  [5980] = {x=869.314, y=-99.781, z=66, rx=180, rz=144.218, shoulder=lefty, elbow=epositive, wrist=wpositive, fatherId=fReference[0]}
  [5981] = {x=870.574, y=-98.873, z=66, rx=180, rz=144.172, shoulder=lefty, elbow=epositive, wrist=wpositive, fatherId=fReference[0]}
  [5982] = {x=871.834, y=-97.963, z=66, rx=-180, rz=144.126, shoulder=lefty, elbow=epositive, wrist=wpositive, fatherId=fReference[0]}
  [5983] = {x=873.094, y=-97.052, z=66, rx=-180, rz=144.08, shoulder=lefty, elbow=epositive, wrist=wpositive, fatherId=fReference[0]}
  [5984] = {x=874.353, y=-96.14, z=66, rx=180, rz=144.036, shoulder=lefty, elbow=epositive, wrist=wpositive, fatherId=fReference[0]}
  [5985] = {x=875.611, y=-95.227, z=66, rx=-180, rz=143.991, shoulder=lefty, elbow=epositive, wrist=wpositive, fatherId=fReference[0]}
  [5986] = {x=876.869, y=-94.313, z=66, rx=180, rz=143.947, shoulder=lefty, elbow=epositive, wrist=wpositive, fatherId=fReference[0]}
  [5987] = {x=878.127, y=-93.397, z=66, rx=180, rz=143.904, shoulder=lefty, elbow=epositive, wrist=wpositive, fatherId=fReference[0]}
  [5988] = {x=879.384, y=-92.481, z=66, rx=180, rz=143.861, shoulder=lefty, elbow=epositive, wrist=wpositive, fatherId=fReference[0]}
  [5989] = {x=880.641, y=-91.563, z=66, rx=-180, rz=143.819, shoulder=lefty, elbow=epositive, wrist=wpositive, fatherId=fReference[0]}
  [5990] = {x=881.897, y=-90.644, z=66, rx=180, rz=143.777, shoulder=lefty, elbow=epositive, wrist=wpositive, fatherId=fReference[0]}
  [5991] = {x=883.153, y=-89.724, z=66, rx=-180, rz=143.735, shoulder=lefty, elbow=epositive, wrist=wpositive, fatherId=fReference[0]}
  [5992] = {x=884.409, y=-88.803, z=66, rx=-180, rz=143.694, shoulder=lefty, elbow=epositive, wrist=wpositive, fatherId=fReference[0]}
  [5993] = {x=885.664, y=-87.881, z=66, rx=-180, rz=143.654, shoulder=lefty, elbow=epositive, wrist=wpositive, fatherId=fReference[0]}
  [5994] = {x=886.919, y=-86.957, z=66, rx=180, rz=143.614, shoulder=lefty, elbow=epositive, wrist=wpositive, fatherId=fReference[0]}
  [5995] = {x=888.173, y=-86.033, z=66, rx=180, rz=143.574, shoulder=lefty, elbow=epositive, wrist=wpositive, fatherId=fReference[0]}
  [5996] = {x=889.427, y=-85.108, z=66, rx=180, rz=143.535, shoulder=lefty, elbow=epositive, wrist=wpositive, fatherId=fReference[0]}
  [5997] = {x=890.681, y=-84.181, z=66, rx=180, rz=143.497, shoulder=lefty, elbow=epositive, wrist=wpositive, fatherId=fReference[0]}
  [5998] = {x=891.934, y=-83.254, z=66, rx=-180, rz=143.459, shoulder=lefty, elbow=epositive, wrist=wpositive, fatherId=fReference[0]}
  [5999] = {x=893.187, y=-82.325, z=66, rx=-180, rz=143.421, shoulder=lefty, elbow=epositive, wrist=wpositive, fatherId=fReference[0]}
  [6000] = {x=894.439, y=-81.396, z=66, rx=180, rz=143.384, shoulder=lefty, elbow=epositive, wrist=wpositive, fatherId=fReference[0]}
  [6001] = {x=895.691, y=-80.465, z=66, rx=180, rz=143.347, shoulder=lefty, elbow=epositive, wrist=wpositive, fatherId=fReference[0]}
  [6002] = {x=896.943, y=-79.534, z=66, rx=-180, rz=143.311, shoulder=lefty, elbow=epositive, wrist=wpositive, fatherId=fReference[0]}
  [6003] = {x=898.195, y=-78.602, z=66, rx=180, rz=143.275, shoulder=lefty, elbow=epositive, wrist=wpositive, fatherId=fReference[0]}
  [6004] = {x=899.446, y=-77.668, z=66, rx=-180, rz=143.24, shoulder=lefty, elbow=epositive, wrist=wpositive, fatherId=fReference[0]}
  [6005] = {x=900.696, y=-76.734, z=66, rx=-180, rz=143.205, shoulder=lefty, elbow=epositive, wrist=wpositive, fatherId=fReference[0]}
  [6006] = {x=901.947, y=-75.799, z=66, rx=-180, rz=143.171, shoulder=lefty, elbow=epositive, wrist=wpositive, fatherId=fReference[0]}
  [6007] = {x=903.197, y=-74.862, z=66, rx=180, rz=143.137, shoulder=lefty, elbow=epositive, wrist=wpositive, fatherId=fReference[0]}
  [6008] = {x=904.447, y=-73.925, z=66, rx=180, rz=143.103, shoulder=lefty, elbow=epositive, wrist=wpositive, fatherId=fReference[0]}
  [6009] = {x=905.696, y=-72.987, z=66, rx=180, rz=143.07, shoulder=lefty, elbow=epositive, wrist=wpositive, fatherId=fReference[0]}
  [6010] = {x=906.945, y=-72.049, z=66, rx=180, rz=143.038, shoulder=lefty, elbow=epositive, wrist=wpositive, fatherId=fReference[0]}
  [6011] = {x=908.194, y=-71.109, z=66, rx=-180, rz=143.006, shoulder=lefty, elbow=epositive, wrist=wpositive, fatherId=fReference[0]}
  [6012] = {x=909.442, y=-70.168, z=66, rx=-180, rz=142.974, shoulder=lefty, elbow=epositive, wrist=wpositive, fatherId=fReference[0]}
  [6013] = {x=910.69, y=-69.227, z=66, rx=180, rz=142.943, shoulder=lefty, elbow=epositive, wrist=wpositive, fatherId=fReference[0]}
  [6014] = {x=911.938, y=-68.285, z=66, rx=-180, rz=142.912, shoulder=lefty, elbow=epositive, wrist=wpositive, fatherId=fReference[0]}
  [6015] = {x=913.185, y=-67.342, z=66, rx=180, rz=142.882, shoulder=lefty, elbow=epositive, wrist=wpositive, fatherId=fReference[0]}
  [6016] = {x=914.433, y=-66.398, z=66, rx=-180, rz=142.853, shoulder=lefty, elbow=epositive, wrist=wpositive, fatherId=fReference[0]}
  [6017] = {x=915.68, y=-65.453, z=66, rx=180, rz=142.823, shoulder=lefty, elbow=epositive, wrist=wpositive, fatherId=fReference[0]}
  [6018] = {x=916.926, y=-64.508, z=66, rx=180, rz=142.794, shoulder=lefty, elbow=epositive, wrist=wpositive, fatherId=fReference[0]}
  [6019] = {x=918.172, y=-63.562, z=66, rx=-180, rz=142.766, shoulder=lefty, elbow=epositive, wrist=wpositive, fatherId=fReference[0]}
  [6020] = {x=919.418, y=-62.615, z=66, rx=-180, rz=142.738, shoulder=lefty, elbow=epositive, wrist=wpositive, fatherId=fReference[0]}
  [6021] = {x=920.664, y=-61.667, z=66, rx=180, rz=142.71, shoulder=lefty, elbow=epositive, wrist=wpositive, fatherId=fReference[0]}
  [6022] = {x=921.91, y=-60.719, z=66, rx=180, rz=142.683, shoulder=lefty, elbow=epositive, wrist=wpositive, fatherId=fReference[0]}
  [6023] = {x=923.155, y=-59.769, z=66, rx=-180, rz=142.657, shoulder=lefty, elbow=epositive, wrist=wpositive, fatherId=fReference[0]}
  [6024] = {x=924.4, y=-58.82, z=66, rx=180, rz=142.631, shoulder=lefty, elbow=epositive, wrist=wpositive, fatherId=fReference[0]}
  [6025] = {x=925.644, y=-57.869, z=66, rx=180, rz=142.605, shoulder=lefty, elbow=epositive, wrist=wpositive, fatherId=fReference[0]}
  [6026] = {x=926.889, y=-56.918, z=66, rx=180, rz=142.58, shoulder=lefty, elbow=epositive, wrist=wpositive, fatherId=fReference[0]}
  [6027] = {x=928.133, y=-55.966, z=66, rx=-180, rz=142.555, shoulder=lefty, elbow=epositive, wrist=wpositive, fatherId=fReference[0]}
  [6028] = {x=929.377, y=-55.013, z=66, rx=-180, rz=142.53, shoulder=lefty, elbow=epositive, wrist=wpositive, fatherId=fReference[0]}
  [6029] = {x=930.621, y=-54.06, z=66, rx=180, rz=142.507, shoulder=lefty, elbow=epositive, wrist=wpositive, fatherId=fReference[0]}
  [6030] = {x=931.864, y=-53.106, z=66, rx=180, rz=142.483, shoulder=lefty, elbow=epositive, wrist=wpositive, fatherId=fReference[0]}
  [6031] = {x=933.107, y=-52.152, z=66, rx=180, rz=142.46, shoulder=lefty, elbow=epositive, wrist=wpositive, fatherId=fReference[0]}
  [6032] = {x=934.35, y=-51.197, z=66, rx=-180, rz=142.437, shoulder=lefty, elbow=epositive, wrist=wpositive, fatherId=fReference[0]}
  [6033] = {x=935.593, y=-50.241, z=66, rx=-180, rz=142.415, shoulder=lefty, elbow=epositive, wrist=wpositive, fatherId=fReference[0]}
  [6034] = {x=936.835, y=-49.284, z=66, rx=-180, rz=142.393, shoulder=lefty, elbow=epositive, wrist=wpositive, fatherId=fReference[0]}
  [6035] = {x=938.078, y=-48.328, z=66, rx=-180, rz=142.372, shoulder=lefty, elbow=epositive, wrist=wpositive, fatherId=fReference[0]}
  [6036] = {x=939.32, y=-47.37, z=66, rx=-180, rz=142.351, shoulder=lefty, elbow=epositive, wrist=wpositive, fatherId=fReference[0]}
  [6037] = {x=940.561, y=-46.412, z=66, rx=180, rz=142.331, shoulder=lefty, elbow=epositive, wrist=wpositive, fatherId=fReference[0]}
  [6038] = {x=941.803, y=-45.454, z=66, rx=180, rz=142.311, shoulder=lefty, elbow=epositive, wrist=wpositive, fatherId=fReference[0]}
  [6039] = {x=943.044, y=-44.494, z=66, rx=180, rz=142.291, shoulder=lefty, elbow=epositive, wrist=wpositive, fatherId=fReference[0]}
  [6040] = {x=944.286, y=-43.535, z=66, rx=180, rz=142.272, shoulder=lefty, elbow=epositive, wrist=wpositive, fatherId=fReference[0]}
  [6041] = {x=945.527, y=-42.575, z=66, rx=-180, rz=142.254, shoulder=lefty, elbow=epositive, wrist=wpositive, fatherId=fReference[0]}
  [6042] = {x=946.768, y=-41.614, z=66, rx=180, rz=142.235, shoulder=lefty, elbow=epositive, wrist=wpositive, fatherId=fReference[0]}
  [6043] = {x=948.008, y=-40.653, z=66, rx=180, rz=142.217, shoulder=lefty, elbow=epositive, wrist=wpositive, fatherId=fReference[0]}
  [6044] = {x=949.249, y=-39.691, z=66, rx=-180, rz=142.2, shoulder=lefty, elbow=epositive, wrist=wpositive, fatherId=fReference[0]}
  [6045] = {x=950.489, y=-38.729, z=66, rx=180, rz=142.183, shoulder=lefty, elbow=epositive, wrist=wpositive, fatherId=fReference[0]}
  [6046] = {x=951.729, y=-37.767, z=66, rx=-180, rz=142.167, shoulder=lefty, elbow=epositive, wrist=wpositive, fatherId=fReference[0]}
  [6047] = {x=952.969, y=-36.804, z=66, rx=180, rz=142.151, shoulder=lefty, elbow=epositive, wrist=wpositive, fatherId=fReference[0]}
  [6048] = {x=954.209, y=-35.841, z=66, rx=-180, rz=142.135, shoulder=lefty, elbow=epositive, wrist=wpositive, fatherId=fReference[0]}
  [6049] = {x=955.448, y=-34.877, z=66, rx=180, rz=142.12, shoulder=lefty, elbow=epositive, wrist=wpositive, fatherId=fReference[0]}
  [6050] = {x=956.688, y=-33.913, z=66, rx=180, rz=142.105, shoulder=lefty, elbow=epositive, wrist=wpositive, fatherId=fReference[0]}
  [6051] = {x=957.927, y=-32.948, z=66, rx=-180, rz=142.09, shoulder=lefty, elbow=epositive, wrist=wpositive, fatherId=fReference[0]}
  [6052] = {x=959.166, y=-31.983, z=66, rx=-180, rz=142.076, shoulder=lefty, elbow=epositive, wrist=wpositive, fatherId=fReference[0]}
  [6053] = {x=960.405, y=-31.018, z=66, rx=-180, rz=142.063, shoulder=lefty, elbow=epositive, wrist=wpositive, fatherId=fReference[0]}
  [6054] = {x=961.644, y=-30.052, z=66, rx=180, rz=142.05, shoulder=lefty, elbow=epositive, wrist=wpositive, fatherId=fReference[0]}
  [6055] = {x=962.882, y=-29.086, z=66, rx=180, rz=142.037, shoulder=lefty, elbow=epositive, wrist=wpositive, fatherId=fReference[0]}
  [6056] = {x=964.121, y=-28.12, z=66, rx=180, rz=142.025, shoulder=lefty, elbow=epositive, wrist=wpositive, fatherId=fReference[0]}
  [6057] = {x=965.359, y=-27.153, z=66, rx=-180, rz=142.013, shoulder=lefty, elbow=epositive, wrist=wpositive, fatherId=fReference[0]}
  [6058] = {x=966.598, y=-26.186, z=66, rx=180, rz=142.002, shoulder=lefty, elbow=epositive, wrist=wpositive, fatherId=fReference[0]}
  [6059] = {x=967.836, y=-25.219, z=66, rx=-180, rz=141.991, shoulder=lefty, elbow=epositive, wrist=wpositive, fatherId=fReference[0]}
  [6060] = {x=969.074, y=-24.251, z=66, rx=-180, rz=141.98, shoulder=lefty, elbow=epositive, wrist=wpositive, fatherId=fReference[0]}
  [6061] = {x=970.312, y=-23.283, z=66, rx=180, rz=141.97, shoulder=lefty, elbow=epositive, wrist=wpositive, fatherId=fReference[0]}
  [6062] = {x=971.55, y=-22.315, z=66, rx=180, rz=141.96, shoulder=lefty, elbow=epositive, wrist=wpositive, fatherId=fReference[0]}
  [6063] = {x=972.787, y=-21.347, z=66, rx=180, rz=141.951, shoulder=lefty, elbow=epositive, wrist=wpositive, fatherId=fReference[0]}
  [6064] = {x=974.025, y=-20.378, z=66, rx=-180, rz=141.942, shoulder=lefty, elbow=epositive, wrist=wpositive, fatherId=fReference[0]}
  [6065] = {x=975.263, y=-19.409, z=66, rx=180, rz=141.934, shoulder=lefty, elbow=epositive, wrist=wpositive, fatherId=fReference[0]}
  [6066] = {x=976.5, y=-18.44, z=66, rx=180, rz=141.926, shoulder=lefty, elbow=epositive, wrist=wpositive, fatherId=fReference[0]}
  [6067] = {x=977.737, y=-17.471, z=66, rx=180, rz=141.918, shoulder=lefty, elbow=epositive, wrist=wpositive, fatherId=fReference[0]}
  [6068] = {x=978.975, y=-16.501, z=66, rx=-180, rz=141.911, shoulder=lefty, elbow=epositive, wrist=wpositive, fatherId=fReference[0]}
  [6069] = {x=980.212, y=-15.532, z=66, rx=180, rz=141.904, shoulder=lefty, elbow=epositive, wrist=wpositive, fatherId=fReference[0]}
  [6070] = {x=981.449, y=-14.562, z=66, rx=-180, rz=141.898, shoulder=lefty, elbow=epositive, wrist=wpositive, fatherId=fReference[0]}
  [6071] = {x=982.686, y=-13.592, z=66, rx=-180, rz=141.892, shoulder=lefty, elbow=epositive, wrist=wpositive, fatherId=fReference[0]}
  [6072] = {x=983.923, y=-12.621, z=66, rx=180, rz=141.887, shoulder=lefty, elbow=epositive, wrist=wpositive, fatherId=fReference[0]}
  [6073] = {x=985.16, y=-11.651, z=66, rx=-180, rz=141.882, shoulder=lefty, elbow=epositive, wrist=wpositive, fatherId=fReference[0]}
  [6074] = {x=986.397, y=-10.681, z=66, rx=-180, rz=141.877, shoulder=lefty, elbow=epositive, wrist=wpositive, fatherId=fReference[0]}
  [6075] = {x=987.634, y=-9.71, z=66, rx=180, rz=141.873, shoulder=lefty, elbow=epositive, wrist=wpositive, fatherId=fReference[0]}
  [6076] = {x=988.87, y=-8.739, z=66, rx=-180, rz=141.869, shoulder=lefty, elbow=epositive, wrist=wpositive, fatherId=fReference[0]}
  [6077] = {x=990.107, y=-7.769, z=66, rx=180, rz=141.866, shoulder=lefty, elbow=epositive, wrist=wpositive, fatherId=fReference[0]}
  [6078] = {x=991.344, y=-6.798, z=66, rx=180, rz=141.863, shoulder=lefty, elbow=epositive, wrist=wpositive, fatherId=fReference[0]}
  [6079] = {x=992.58, y=-5.827, z=66, rx=-180, rz=141.86, shoulder=lefty, elbow=epositive, wrist=wpositive, fatherId=fReference[0]}
  [6080] = {x=993.817, y=-4.856, z=66, rx=180, rz=141.858, shoulder=lefty, elbow=epositive, wrist=wpositive, fatherId=fReference[0]}
  [6081] = {x=995.054, y=-3.885, z=66, rx=180, rz=141.857, shoulder=lefty, elbow=epositive, wrist=wpositive, fatherId=fReference[0]}
  [6082] = {x=996.29, y=-2.914, z=66, rx=-180, rz=141.855, shoulder=lefty, elbow=epositive, wrist=wpositive, fatherId=fReference[0]}
  [6083] = {x=997.527, y=-1.942, z=66, rx=180, rz=141.854, shoulder=lefty, elbow=epositive, wrist=wpositive, fatherId=fReference[0]}
  [6084] = {x=998.763, y=-0.971, z=66, rx=180, rz=141.854, shoulder=lefty, elbow=epositive, wrist=wpositive, fatherId=fReference[0]}
  [6085] = {x=1000, z=66, rx=180, rz=141.854, shoulder=lefty, elbow=epositive, wrist=wpositive, fatherId=fReference[0]}
  [6086] = {x=1000, z=66, rx=180, rz=141.854, shoulder=lefty, elbow=epositive, wrist=wpositive, fatherId=fReference[0]}
  [6087] = {x=1000, z=166, rx=180, rz=141.854, shoulder=lefty, elbow=epositive, wrist=wpositive, fatherId=fReference[0]}
public tool tTool = {z=600, rz=55, fatherId=flange[0], ioLink=valve1}
public num kk
public bool spd_cntl
public mdesc cnst_vel = {tmax=100, rmax=100, leave=0.1, reach=0.1, blend=cartesian}
public jointRx Jnt_cnfg = {j3=90, j5=90, j6=90}
public num Ref_Vel
sio sioASCII = {link=Socket\trsf_sv}
public bool check_status
aio Tpompe = {link=CanIO\RemIO\remio0_QW}
dio doValve1 = {link=valve1}
dio doValve2 = {link=valve2}
